TYPE ST_MTI_INPUT :
STRUCT
  EventState            : BIT;
  EventTime             : UDINT;
END_STRUCT
END_TYPE

(* stored: Version 1.1.0.1, ProductVersion 3.1.4024.12
   DUT ST_MTI_INPUT: Id {f817458e-2c0d-4ada-932c-6a2afaabdd2d} *)
